{attribute 'qualified_only'}
{attribute 'to_string'}
{attribute 'strict'}
TYPE E_CONFIG_CTRL :
(
  NO_INIT,
	IDLE,

  READ  := 20,
  WRITE := 30
)UINT;
END_TYPE

(* stored: Version 1.1.0.1, ProductVersion 3.1.4024.13
   DUT E_CONFIG_CTRL: Id {9bb3bef8-211a-49fb-81fa-53bbdf984366} *)
